(* Logix 5000 project; controller RG_Chopper vendor 1 type 14 code 235 rev 32.12; software revision 32.04; part 6 of 6 *)
(* tags used below, declared in another part *)
   ALARM_S_FATAL : BOOL;   // Fatal Alarm Safety Map Stops All Operation
   DBX101_S_START : BOOL;   // DBX-101 Safety map Agitator Start
   DBX102B_S_En : BOOL;   // DBX-102 Drive Safety Enable
   DBX103_S_START : BOOL;   // DBX-103 Safety map Hot Water Pump Start
   Flash_S : BOOL;   // Safety Flash Bit
   KR101_DUMPER_PERM : BOOL;   // Dumper Permissive NON-FATAL ALARM 0 = ALARM
   M104S_DWN_CTL : CONFIGURABLE_ROUT;   // DBX-104 Dump Elevator Safety Starter Down Output
   M104S_STRT_CTL : CONFIGURABLE_ROUT;   // DBX-104 Dump Elevator Safety Starter Enable Output
   M104S_UP_CTL : CONFIGURABLE_ROUT;   // DBX-104 Dump Elevator Safety Starter UP Output
   S_HORN : BOOL;   // Audible Alarm HORN
   S_TMR_1 : TIMER;   // Safety Timer #1
   S_TMR_2 : TIMER;   // Safety Timer #2
   SCRL_STRT : TIMER;   // Scroll Startup Warning Timer
(* SafetyProgram, continued *)

ROUTINE OutLink   (* ladder *)
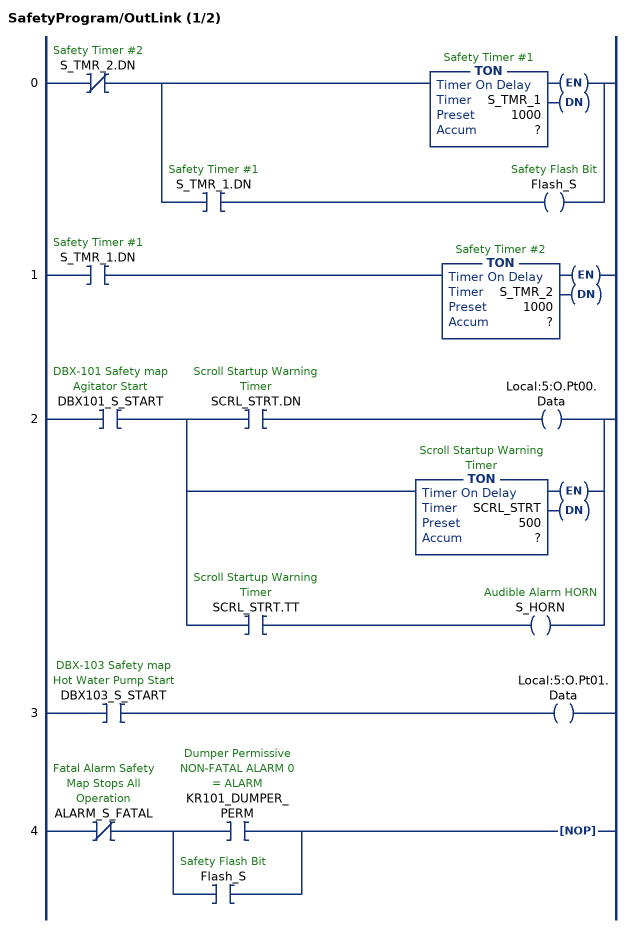
   0: XIO(S_TMR_2.DN)[TON(S_TMR_1,?,?) ,XIC(S_TMR_1.DN) OTE(Flash_S) ];
   1: XIC(S_TMR_1.DN)TON(S_TMR_2,?,?);
   2: XIC(DBX101_S_START)[XIC(SCRL_STRT.DN) OTE(Local:5:O.Pt00.Data) ,TON(SCRL_STRT,?,?) ,XIC(SCRL_STRT.TT) OTE(S_HORN) ];
   3: XIC(DBX103_S_START)OTE(Local:5:O.Pt01.Data);
   4: XIO(ALARM_S_FATAL)[XIC(KR101_DUMPER_PERM) ,XIC(Flash_S) ]NOP();
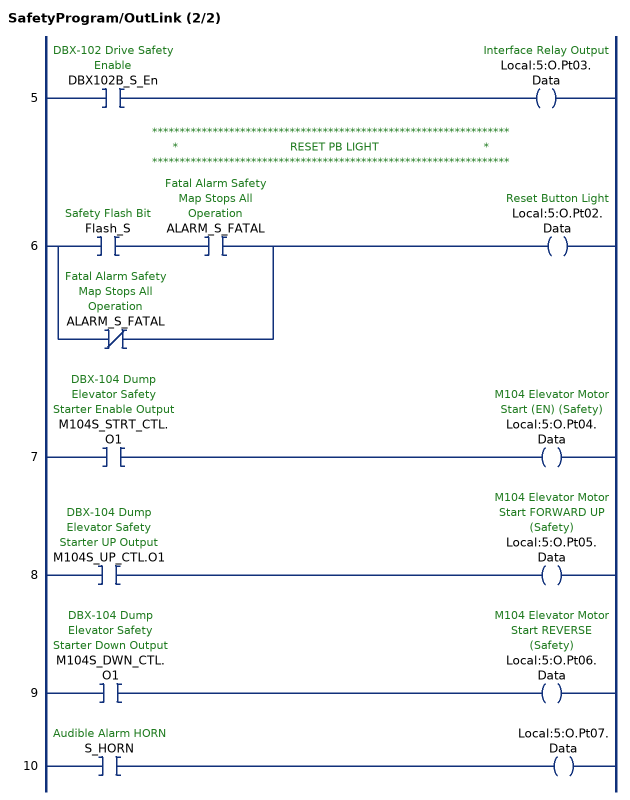
   5: XIC(DBX102B_S_En)OTE(Local:5:O.Pt03.Data);
   // *****************************************************************
   // *                                RESET PB LIGHT                              *
   // *****************************************************************
   6: [XIC(Flash_S) XIC(ALARM_S_FATAL) ,XIO(ALARM_S_FATAL) ]OTE(Local:5:O.Pt02.Data);
   7: XIC(M104S_STRT_CTL.O1)OTE(Local:5:O.Pt04.Data);
   8: XIC(M104S_UP_CTL.O1)OTE(Local:5:O.Pt05.Data);
   9: XIC(M104S_DWN_CTL.O1)OTE(Local:5:O.Pt06.Data);
   10: XIC(S_HORN)OTE(Local:5:O.Pt07.Data);
END_ROUTINE
END_PROGRAM
